FUNCTION_BLOCK FB_NCI
VAR_INPUT
END_VAR
VAR_OUTPUT
END_VAR
VAR
END_VAR

END_FUNCTION_BLOCK

(* stored: Version 1.1.0.1, ProductVersion 3.1.4024.12
   POU FB_NCI: Id {a10e90fe-73ba-4e2b-a9a5-81d463ea7a9b}, SpecialFunc None *)
